INTERFACE ILog

METHOD SetLogger : BOOL
VAR_INPUT
    ref2Core : ILogCore;
END_VAR
END_METHOD

END_INTERFACE

(* stored: Version 1.1.0.1
   Itf ILog: Id {412ad8b8-57e1-419f-af21-e16e50d36d6b}
   Method SetLogger: Id {d997efda-3f08-4614-802a-e86242c0eb02} *)
